// A watchdog function block. Observer "variable" input - if the value does not change within the "timeout" parameter, status will return "FALSE"
FUNCTION_BLOCK FB_Watchdog
VAR_INPUT
	variable	: BOOL;	// Variable to observe
	timeout		: TIME;	// Time within the variable needs to change it's state before status is reported as FALSE
END_VAR

VAR_OUTPUT
	status	: BOOL;	// TRUE = OK, FALSE = timeout
END_VAR

VAR
	Ton_TrueTimer	: Tc2_Standard.TON;
	Ton_Falsetimer	: Tc2_Standard.TON;
END_VAR

Ton_TrueTimer(IN := variable, PT := timeout);
Ton_Falsetimer(IN := NOT variable, PT := timeout);


status := Ton_TrueTimer.Q = FALSE AND  Ton_Falsetimer.Q = FALSE;

END_FUNCTION_BLOCK

(* stored: Version 1.1.0.1, ProductVersion 3.1.4024.15
   POU FB_Watchdog: Id {110d80c9-88e3-070c-2af5-b43c21617595}, SpecialFunc None *)
